FUNCTION_BLOCK SPINDLE_SPEED (* Converts spindle speed and sends it *)
  (* Standard: 61499-2 *)
  (* Version 1.0, 09-01-12, Guilherme Jarentchuk, Universidade do Estado de Santa Catarina *)
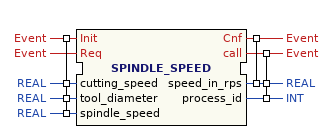
  EVENT_INPUT
    Init WITH cutting_speed, tool_diameter, spindle_speed; (* Initialize execution *)
    Req; (* Request to finish *)
  END_EVENT
  EVENT_OUTPUT
    Cnf WITH speed_in_rps; (* Confirm execution *)
    call WITH speed_in_rps, process_id; (* Call execution device *)
  END_EVENT
  VAR_INPUT
    cutting_speed : REAL; (* Spindle speed in m/s *)
    tool_diameter : REAL; (* In mm *)
    spindle_speed : REAL; (* In rot/s *)
  END_VAR
  VAR_OUTPUT
    speed_in_rps : REAL;
    process_id : INT;
  END_VAR
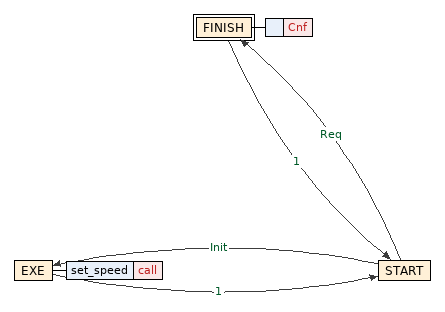
  EC_STATES
    FINISH : -> Cnf;
    START;
    EXE : set_speed -> call;
  END_STATES
  EC_TRANSITIONS
    FINISH TO START := 1;
    START TO EXE := Init;
    START TO FINISH := Req;
    EXE TO START := 1;
  END_TRANSITIONS
  ALGORITHM set_speed IN Lua:
if( spindle_speed > 0 ) then
	speed_in_rps = spindle_speed
elseif( cutting_speed > 0) and ( tool_diameter > 0 ) then
	speed_in_rps = cutting_speed/( (tool_diameter/1000)*math.pi )
end
process_id = -5
  END_ALGORITHM
END_FUNCTION_BLOCK
